TYPE U_OdriveDwordBytes :
UNION
    Value : DWORD;
    Bytes : ARRAY[0..3] OF BYTE;
END_UNION
END_TYPE

(* stored: Version 1.1.0.1
   DUT U_OdriveDwordBytes: Id {22FE0B43-EC16-452D-A3A8-EA2DD30F0B1E} *)
